(* IEC 61131-3 sources: AXOpen/src/components.festo.drives/app/src/IO, 10 files *)

(* ---- HwIdentifiers.st ---- *)
TYPE
	HwIdentifiers : ULINT
	(
		PLC_LINE_Rail_0 :=	ULINT#256,
		PLC_LINE_PLC_LINE :=	ULINT#48,
		PLC_LINE_Card_reader_writer_1 :=	ULINT#51,
		PLC_LINE_CPU_display_1 :=	ULINT#54,
		PLC_LINE_OPC_UA_1 :=	ULINT#117,
		PLC_LINE_PROFINET_interface_1 :=	ULINT#64,
		PLC_LINE_Port_1 :=	ULINT#65,
		PLC_LINE_Port_2 :=	ULINT#66,
		PLC_LINE_PROFINET_interface_2 :=	ULINT#72,
		PLC_LINE_DP_interface_1 :=	ULINT#60,
		PLC_LINE_PROFINET_interface_GBIT_3 :=	ULINT#120,
		ST3_indradrive_Rack :=	ULINT#336,
		ST3_indradrive_ST3_indradrive :=	ULINT#337,
		ST3_indradrive_PN_IO :=	ULINT#338,
		ST3_indradrive_Port_1_RJ45 :=	ULINT#339,
		ST3_indradrive_Port_2_RJ45 :=	ULINT#340,
		ST3_indradrive_DAP_1 :=	ULINT#341,
		ST3_indradrive_ID_FMod_NotUsed :=	ULINT#342,
		ST3_indradrive_ID_PaCh_5Words :=	ULINT#258,
		ST3_indradrive_ID_InMod_9Words :=	ULINT#262,
		ST3_indradrive_ID_OutMod_13Words :=	ULINT#259,
		cmmtas_PN_IO_Interface :=	ULINT#271,
		cmmtas_Port_1 :=	ULINT#260,
		cmmtas_Port_2 :=	ULINT#261,
		cmmtas_CMMT_AS_MP :=	ULINT#272,
		cmmtas_Module_Access_Point :=	ULINT#264,
		cmmtas_Siemens_telegram_111_PZD_12_12 :=	ULINT#265,
		cmmtas_Siemens_telegram_750_PZD_4_1 :=	ULINT#266,
		NONE:= ULINT#0
	);
END_TYPE

(* ---- HwInputs.st ---- *)
TYPE
	HwInputs : STRUCT
		ST3_indradrive_ID_PaCh_5Words AT %B10 : ARRAY[0..9] OF BYTE;
		ST3_indradrive_ID_InMod_9Words AT %B20 : ARRAY[0..17] OF BYTE;
		cmmtas_DO_SERVO_1_Siemens_telegram_111_PZD_12_12 AT %B100 : ARRAY[0..23] OF BYTE;
		cmmtas_DO_SERVO_1_Siemens_telegram_750_PZD_4_1 AT %B124 : WORD;
	END_STRUCT;
END_TYPE

(* ---- HwOutputs.st ---- *)
TYPE
	HwOutputs : STRUCT
		ST3_indradrive_ID_PaCh_5Words AT %B10 : ARRAY[0..9] OF BYTE;
		ST3_indradrive_ID_OutMod_13Words AT %B20 : ARRAY[0..25] OF BYTE;
		cmmtas_DO_SERVO_1_Siemens_telegram_111_PZD_12_12 AT %B100 : ARRAY[0..23] OF BYTE;
		cmmtas_DO_SERVO_1_Siemens_telegram_750_PZD_4_1 AT %B124 : ARRAY[0..7] OF BYTE;
	END_STRUCT;
END_TYPE

(* ---- Inputs.st ---- *)
NAMESPACE AXOpen.Components.Festo.Drives
    TYPE
        {S7.extern=ReadWrite}
        {#ix-attr:[Container(Layout.Wrap)]}
        Inputs : STRUCT
	        // Module festo_cmmtas/DoServo
	        festo_cmmtas_DoServo_SiemensTelegram111_PZD_12_12_Input AT %B0 : festo_cmmtas_DoServo_SiemensTelegram111_PZD_12_12_Input_Layout;

	        festo_cmmtas_DoServo_SiemensTelegram750_PZD_4_1_Input AT %B24 : festo_cmmtas_DoServo_SiemensTelegram750_PZD_4_1_Input_Layout;

        END_STRUCT;
    END_TYPE
END_NAMESPACE

(* ---- IoStructures.st ---- *)
NAMESPACE AXOpen.Components.Festo.Drives
	TYPE
        {S7.extern=ReadWrite}
        {#ix-attr:[Container(Layout.Wrap)]}
	    festo_cmmtas_DoServo_SiemensTelegram111_PZD_12_12_Input_Layout : STRUCT
	        Signals_0 AT %X0.0 : BOOL;
	        Signals_1 AT %X0.1 : BOOL;
	        Signals_2 AT %X0.2 : BOOL;
	        Signals_3 AT %X0.3 : BOOL;
	        Signals_4 AT %X0.4 : BOOL;
	        Signals_5 AT %X0.5 : BOOL;
	        Signals_6 AT %X0.6 : BOOL;
	        Signals_7 AT %X0.7 : BOOL;
	        Signals_8 AT %X1.0 : BOOL;
	        Signals_9 AT %X1.1 : BOOL;
	        Signals_10 AT %X1.2 : BOOL;
	        Signals_11 AT %X1.3 : BOOL;
	        Signals_12 AT %X1.4 : BOOL;
	        Signals_13 AT %X1.5 : BOOL;
	        Signals_14 AT %X1.6 : BOOL;
	        Signals_15 AT %X1.7 : BOOL;
	        Signals_16 AT %X2.0 : BOOL;
	        Signals_17 AT %X2.1 : BOOL;
	        Signals_18 AT %X2.2 : BOOL;
	        Signals_19 AT %X2.3 : BOOL;
	        Signals_20 AT %X2.4 : BOOL;
	        Signals_21 AT %X2.5 : BOOL;
	        Signals_22 AT %X2.6 : BOOL;
	        Signals_23 AT %X2.7 : BOOL;
	        Signals_24 AT %X3.0 : BOOL;
	        Signals_25 AT %X3.1 : BOOL;
	        Signals_26 AT %X3.2 : BOOL;
	        Signals_27 AT %X3.3 : BOOL;
	        Signals_28 AT %X3.4 : BOOL;
	        Signals_29 AT %X3.5 : BOOL;
	        Signals_30 AT %X3.6 : BOOL;
	        Signals_31 AT %X3.7 : BOOL;
	        Signals_32 AT %X4.0 : BOOL;
	        Signals_33 AT %X4.1 : BOOL;
	        Signals_34 AT %X4.2 : BOOL;
	        Signals_35 AT %X4.3 : BOOL;
	        Signals_36 AT %X4.4 : BOOL;
	        Signals_37 AT %X4.5 : BOOL;
	        Signals_38 AT %X4.6 : BOOL;
	        Signals_39 AT %X4.7 : BOOL;
	        Signals_40 AT %X5.0 : BOOL;
	        Signals_41 AT %X5.1 : BOOL;
	        Signals_42 AT %X5.2 : BOOL;
	        Signals_43 AT %X5.3 : BOOL;
	        Signals_44 AT %X5.4 : BOOL;
	        Signals_45 AT %X5.5 : BOOL;
	        Signals_46 AT %X5.6 : BOOL;
	        Signals_47 AT %X5.7 : BOOL;
	        Signals_48 AT %X6.0 : BOOL;
	        Signals_49 AT %X6.1 : BOOL;
	        Signals_50 AT %X6.2 : BOOL;
	        Signals_51 AT %X6.3 : BOOL;
	        Signals_52 AT %X6.4 : BOOL;
	        Signals_53 AT %X6.5 : BOOL;
	        Signals_54 AT %X6.6 : BOOL;
	        Signals_55 AT %X6.7 : BOOL;
	        Signals_56 AT %X7.0 : BOOL;
	        Signals_57 AT %X7.1 : BOOL;
	        Signals_58 AT %X7.2 : BOOL;
	        Signals_59 AT %X7.3 : BOOL;
	        Signals_60 AT %X7.4 : BOOL;
	        Signals_61 AT %X7.5 : BOOL;
	        Signals_62 AT %X7.6 : BOOL;
	        Signals_63 AT %X7.7 : BOOL;
	        Signals_64 AT %X8.0 : BOOL;
	        Signals_65 AT %X8.1 : BOOL;
	        Signals_66 AT %X8.2 : BOOL;
	        Signals_67 AT %X8.3 : BOOL;
	        Signals_68 AT %X8.4 : BOOL;
	        Signals_69 AT %X8.5 : BOOL;
	        Signals_70 AT %X8.6 : BOOL;
	        Signals_71 AT %X8.7 : BOOL;
	        Signals_72 AT %X9.0 : BOOL;
	        Signals_73 AT %X9.1 : BOOL;
	        Signals_74 AT %X9.2 : BOOL;
	        Signals_75 AT %X9.3 : BOOL;
	        Signals_76 AT %X9.4 : BOOL;
	        Signals_77 AT %X9.5 : BOOL;
	        Signals_78 AT %X9.6 : BOOL;
	        Signals_79 AT %X9.7 : BOOL;
	        Signals_80 AT %B10 : DWORD;
	        Signals_81 AT %B14 : DWORD;
	        Signals_82 AT %B18 : WORD;
	        Signals_83 AT %B20 : WORD;
	        Signals_84 AT %B22 : WORD;
	    END_STRUCT;
	END_TYPE

	TYPE
        {S7.extern=ReadWrite}
        {#ix-attr:[Container(Layout.Wrap)]}
	    festo_cmmtas_DoServo_SiemensTelegram111_PZD_12_12_Output_Layout : STRUCT
	        Signals_85 AT %X0.0 : BOOL;
	        Signals_86 AT %X0.1 : BOOL;
	        Signals_87 AT %X0.2 : BOOL;
	        Signals_88 AT %X0.3 : BOOL;
	        Signals_89 AT %X0.4 : BOOL;
	        Signals_90 AT %X0.5 : BOOL;
	        Signals_91 AT %X0.6 : BOOL;
	        Signals_92 AT %X0.7 : BOOL;
	        Signals_93 AT %X1.0 : BOOL;
	        Signals_94 AT %X1.1 : BOOL;
	        Signals_95 AT %X1.2 : BOOL;
	        Signals_96 AT %X1.3 : BOOL;
	        Signals_97 AT %X1.4 : BOOL;
	        Signals_98 AT %X1.5 : BOOL;
	        Signals_99 AT %X1.6 : BOOL;
	        Signals_100 AT %X1.7 : BOOL;
	        Signals_101 AT %X2.0 : BOOL;
	        Signals_102 AT %X2.1 : BOOL;
	        Signals_103 AT %X2.2 : BOOL;
	        Signals_104 AT %X2.3 : BOOL;
	        Signals_105 AT %X2.4 : BOOL;
	        Signals_106 AT %X2.5 : BOOL;
	        Signals_107 AT %X2.6 : BOOL;
	        Signals_108 AT %X2.7 : BOOL;
	        Signals_109 AT %X3.0 : BOOL;
	        Signals_110 AT %X3.1 : BOOL;
	        Signals_111 AT %X3.2 : BOOL;
	        Signals_112 AT %X3.3 : BOOL;
	        Signals_113 AT %X3.4 : BOOL;
	        Signals_114 AT %X3.5 : BOOL;
	        Signals_115 AT %X3.6 : BOOL;
	        Signals_116 AT %X3.7 : BOOL;
	        Signals_117 AT %X4.0 : BOOL;
	        Signals_118 AT %X4.1 : BOOL;
	        Signals_119 AT %X4.2 : BOOL;
	        Signals_120 AT %X4.3 : BOOL;
	        Signals_121 AT %X4.4 : BOOL;
	        Signals_122 AT %X4.5 : BOOL;
	        Signals_123 AT %X4.6 : BOOL;
	        Signals_124 AT %X4.7 : BOOL;
	        Signals_125 AT %X5.0 : BOOL;
	        Signals_126 AT %X5.1 : BOOL;
	        Signals_127 AT %X5.2 : BOOL;
	        Signals_128 AT %X5.3 : BOOL;
	        Signals_129 AT %X5.4 : BOOL;
	        Signals_130 AT %X5.5 : BOOL;
	        Signals_131 AT %X5.6 : BOOL;
	        Signals_132 AT %X5.7 : BOOL;
	        Signals_133 AT %X6.0 : BOOL;
	        Signals_134 AT %X6.1 : BOOL;
	        Signals_135 AT %X6.2 : BOOL;
	        Signals_136 AT %X6.3 : BOOL;
	        Signals_137 AT %X6.4 : BOOL;
	        Signals_138 AT %X6.5 : BOOL;
	        Signals_139 AT %X6.6 : BOOL;
	        Signals_140 AT %X6.7 : BOOL;
	        Signals_141 AT %X7.0 : BOOL;
	        Signals_142 AT %X7.1 : BOOL;
	        Signals_143 AT %X7.2 : BOOL;
	        Signals_144 AT %X7.3 : BOOL;
	        Signals_145 AT %X7.4 : BOOL;
	        Signals_146 AT %X7.5 : BOOL;
	        Signals_147 AT %X7.6 : BOOL;
	        Signals_148 AT %X7.7 : BOOL;
	        Signals_149 AT %B8 : WORD;
	        Signals_150 AT %B10 : DINT;
	        Signals_151 AT %B14 : DWORD;
	        Signals_152 AT %B18 : WORD;
	        Signals_153 AT %B20 : WORD;
	        Signals_154 AT %B22 : WORD;
	    END_STRUCT;
	END_TYPE

	TYPE
        {S7.extern=ReadWrite}
        {#ix-attr:[Container(Layout.Wrap)]}
	    festo_cmmtas_DoServo_SiemensTelegram750_PZD_4_1_Input_Layout : STRUCT
	        Signals_0 AT %B0 : WORD;
	    END_STRUCT;
	END_TYPE

	TYPE
        {S7.extern=ReadWrite}
        {#ix-attr:[Container(Layout.Wrap)]}
	    festo_cmmtas_DoServo_SiemensTelegram750_PZD_4_1_Output_Layout : STRUCT
	        Signals_1 AT %B0 : WORD;
	        Signals_2 AT %B2 : WORD;
	        Signals_3 AT %B4 : WORD;
	        Signals_4 AT %B6 : WORD;
	    END_STRUCT;
	END_TYPE
END_NAMESPACE

(* ---- Outputs.st ---- *)
NAMESPACE AXOpen.Components.Festo.Drives
    TYPE
        {S7.extern=ReadWrite}
        {#ix-attr:[Container(Layout.Wrap)]}
        Outputs : STRUCT
            cmmtas_DoServo_Submodule_1_0 AT %B0:  LWORD;
            cmmtas_DoServo_Submodule_1_1 AT %B8:  LWORD;
            cmmtas_DoServo_Submodule_1_2 AT %B16:  LWORD;
            cmmtas_DoServo_Submodule_2 AT %B24:  LWORD;
        END_STRUCT;
    END_TYPE
END_NAMESPACE

(* ---- PlcInputs.st ---- *)
TYPE
	PlcInputs : STRUCT
		ST3_indradrive_ID_PaCh_5Words : ARRAY[0..9] OF BYTE;
		ST3_indradrive_ID_InMod_9Words : ARRAY[0..17] OF BYTE;
		cmmtas_DO_SERVO_1_Siemens_telegram_111_PZD_12_12 : ARRAY[0..23] OF BYTE;
		cmmtas_DO_SERVO_1_Siemens_telegram_750_PZD_4_1 : WORD;
	END_STRUCT;
END_TYPE

(* ---- PlcOutputs.st ---- *)
TYPE
	PlcOutputs : STRUCT
		ST3_indradrive_ID_PaCh_5Words : ARRAY[0..9] OF BYTE;
		ST3_indradrive_ID_OutMod_13Words : ARRAY[0..25] OF BYTE;
		cmmtas_DO_SERVO_1_Siemens_telegram_111_PZD_12_12 : ARRAY[0..23] OF BYTE;
		cmmtas_DO_SERVO_1_Siemens_telegram_750_PZD_4_1 : ARRAY[0..7] OF BYTE;
	END_STRUCT;
END_TYPE

(* ---- CopyInputs.st ---- *)
FUNCTION CopyInputs
	VAR_EXTERNAL
		HwInputs : HwInputs;
		PlcInputs : PlcInputs;
	END_VAR
	PlcInputs.ST3_indradrive_ID_PaCh_5Words[0] := HwInputs.ST3_indradrive_ID_PaCh_5Words[0];
	PlcInputs.ST3_indradrive_ID_PaCh_5Words[1] := HwInputs.ST3_indradrive_ID_PaCh_5Words[1];
	PlcInputs.ST3_indradrive_ID_PaCh_5Words[2] := HwInputs.ST3_indradrive_ID_PaCh_5Words[2];
	PlcInputs.ST3_indradrive_ID_PaCh_5Words[3] := HwInputs.ST3_indradrive_ID_PaCh_5Words[3];
	PlcInputs.ST3_indradrive_ID_PaCh_5Words[4] := HwInputs.ST3_indradrive_ID_PaCh_5Words[4];
	PlcInputs.ST3_indradrive_ID_PaCh_5Words[5] := HwInputs.ST3_indradrive_ID_PaCh_5Words[5];
	PlcInputs.ST3_indradrive_ID_PaCh_5Words[6] := HwInputs.ST3_indradrive_ID_PaCh_5Words[6];
	PlcInputs.ST3_indradrive_ID_PaCh_5Words[7] := HwInputs.ST3_indradrive_ID_PaCh_5Words[7];
	PlcInputs.ST3_indradrive_ID_PaCh_5Words[8] := HwInputs.ST3_indradrive_ID_PaCh_5Words[8];
	PlcInputs.ST3_indradrive_ID_PaCh_5Words[9] := HwInputs.ST3_indradrive_ID_PaCh_5Words[9];
	PlcInputs.ST3_indradrive_ID_InMod_9Words[0] := HwInputs.ST3_indradrive_ID_InMod_9Words[0];
	PlcInputs.ST3_indradrive_ID_InMod_9Words[1] := HwInputs.ST3_indradrive_ID_InMod_9Words[1];
	PlcInputs.ST3_indradrive_ID_InMod_9Words[2] := HwInputs.ST3_indradrive_ID_InMod_9Words[2];
	PlcInputs.ST3_indradrive_ID_InMod_9Words[3] := HwInputs.ST3_indradrive_ID_InMod_9Words[3];
	PlcInputs.ST3_indradrive_ID_InMod_9Words[4] := HwInputs.ST3_indradrive_ID_InMod_9Words[4];
	PlcInputs.ST3_indradrive_ID_InMod_9Words[5] := HwInputs.ST3_indradrive_ID_InMod_9Words[5];
	PlcInputs.ST3_indradrive_ID_InMod_9Words[6] := HwInputs.ST3_indradrive_ID_InMod_9Words[6];
	PlcInputs.ST3_indradrive_ID_InMod_9Words[7] := HwInputs.ST3_indradrive_ID_InMod_9Words[7];
	PlcInputs.ST3_indradrive_ID_InMod_9Words[8] := HwInputs.ST3_indradrive_ID_InMod_9Words[8];
	PlcInputs.ST3_indradrive_ID_InMod_9Words[9] := HwInputs.ST3_indradrive_ID_InMod_9Words[9];
	PlcInputs.ST3_indradrive_ID_InMod_9Words[10] := HwInputs.ST3_indradrive_ID_InMod_9Words[10];
	PlcInputs.ST3_indradrive_ID_InMod_9Words[11] := HwInputs.ST3_indradrive_ID_InMod_9Words[11];
	PlcInputs.ST3_indradrive_ID_InMod_9Words[12] := HwInputs.ST3_indradrive_ID_InMod_9Words[12];
	PlcInputs.ST3_indradrive_ID_InMod_9Words[13] := HwInputs.ST3_indradrive_ID_InMod_9Words[13];
	PlcInputs.ST3_indradrive_ID_InMod_9Words[14] := HwInputs.ST3_indradrive_ID_InMod_9Words[14];
	PlcInputs.ST3_indradrive_ID_InMod_9Words[15] := HwInputs.ST3_indradrive_ID_InMod_9Words[15];
	PlcInputs.ST3_indradrive_ID_InMod_9Words[16] := HwInputs.ST3_indradrive_ID_InMod_9Words[16];
	PlcInputs.ST3_indradrive_ID_InMod_9Words[17] := HwInputs.ST3_indradrive_ID_InMod_9Words[17];
	PlcInputs.cmmtas_DO_SERVO_1_Siemens_telegram_111_PZD_12_12[0] := HwInputs.cmmtas_DO_SERVO_1_Siemens_telegram_111_PZD_12_12[0];
	PlcInputs.cmmtas_DO_SERVO_1_Siemens_telegram_111_PZD_12_12[1] := HwInputs.cmmtas_DO_SERVO_1_Siemens_telegram_111_PZD_12_12[1];
	PlcInputs.cmmtas_DO_SERVO_1_Siemens_telegram_111_PZD_12_12[2] := HwInputs.cmmtas_DO_SERVO_1_Siemens_telegram_111_PZD_12_12[2];
	PlcInputs.cmmtas_DO_SERVO_1_Siemens_telegram_111_PZD_12_12[3] := HwInputs.cmmtas_DO_SERVO_1_Siemens_telegram_111_PZD_12_12[3];
	PlcInputs.cmmtas_DO_SERVO_1_Siemens_telegram_111_PZD_12_12[4] := HwInputs.cmmtas_DO_SERVO_1_Siemens_telegram_111_PZD_12_12[4];
	PlcInputs.cmmtas_DO_SERVO_1_Siemens_telegram_111_PZD_12_12[5] := HwInputs.cmmtas_DO_SERVO_1_Siemens_telegram_111_PZD_12_12[5];
	PlcInputs.cmmtas_DO_SERVO_1_Siemens_telegram_111_PZD_12_12[6] := HwInputs.cmmtas_DO_SERVO_1_Siemens_telegram_111_PZD_12_12[6];
	PlcInputs.cmmtas_DO_SERVO_1_Siemens_telegram_111_PZD_12_12[7] := HwInputs.cmmtas_DO_SERVO_1_Siemens_telegram_111_PZD_12_12[7];
	PlcInputs.cmmtas_DO_SERVO_1_Siemens_telegram_111_PZD_12_12[8] := HwInputs.cmmtas_DO_SERVO_1_Siemens_telegram_111_PZD_12_12[8];
	PlcInputs.cmmtas_DO_SERVO_1_Siemens_telegram_111_PZD_12_12[9] := HwInputs.cmmtas_DO_SERVO_1_Siemens_telegram_111_PZD_12_12[9];
	PlcInputs.cmmtas_DO_SERVO_1_Siemens_telegram_111_PZD_12_12[10] := HwInputs.cmmtas_DO_SERVO_1_Siemens_telegram_111_PZD_12_12[10];
	PlcInputs.cmmtas_DO_SERVO_1_Siemens_telegram_111_PZD_12_12[11] := HwInputs.cmmtas_DO_SERVO_1_Siemens_telegram_111_PZD_12_12[11];
	PlcInputs.cmmtas_DO_SERVO_1_Siemens_telegram_111_PZD_12_12[12] := HwInputs.cmmtas_DO_SERVO_1_Siemens_telegram_111_PZD_12_12[12];
	PlcInputs.cmmtas_DO_SERVO_1_Siemens_telegram_111_PZD_12_12[13] := HwInputs.cmmtas_DO_SERVO_1_Siemens_telegram_111_PZD_12_12[13];
	PlcInputs.cmmtas_DO_SERVO_1_Siemens_telegram_111_PZD_12_12[14] := HwInputs.cmmtas_DO_SERVO_1_Siemens_telegram_111_PZD_12_12[14];
	PlcInputs.cmmtas_DO_SERVO_1_Siemens_telegram_111_PZD_12_12[15] := HwInputs.cmmtas_DO_SERVO_1_Siemens_telegram_111_PZD_12_12[15];
	PlcInputs.cmmtas_DO_SERVO_1_Siemens_telegram_111_PZD_12_12[16] := HwInputs.cmmtas_DO_SERVO_1_Siemens_telegram_111_PZD_12_12[16];
	PlcInputs.cmmtas_DO_SERVO_1_Siemens_telegram_111_PZD_12_12[17] := HwInputs.cmmtas_DO_SERVO_1_Siemens_telegram_111_PZD_12_12[17];
	PlcInputs.cmmtas_DO_SERVO_1_Siemens_telegram_111_PZD_12_12[18] := HwInputs.cmmtas_DO_SERVO_1_Siemens_telegram_111_PZD_12_12[18];
	PlcInputs.cmmtas_DO_SERVO_1_Siemens_telegram_111_PZD_12_12[19] := HwInputs.cmmtas_DO_SERVO_1_Siemens_telegram_111_PZD_12_12[19];
	PlcInputs.cmmtas_DO_SERVO_1_Siemens_telegram_111_PZD_12_12[20] := HwInputs.cmmtas_DO_SERVO_1_Siemens_telegram_111_PZD_12_12[20];
	PlcInputs.cmmtas_DO_SERVO_1_Siemens_telegram_111_PZD_12_12[21] := HwInputs.cmmtas_DO_SERVO_1_Siemens_telegram_111_PZD_12_12[21];
	PlcInputs.cmmtas_DO_SERVO_1_Siemens_telegram_111_PZD_12_12[22] := HwInputs.cmmtas_DO_SERVO_1_Siemens_telegram_111_PZD_12_12[22];
	PlcInputs.cmmtas_DO_SERVO_1_Siemens_telegram_111_PZD_12_12[23] := HwInputs.cmmtas_DO_SERVO_1_Siemens_telegram_111_PZD_12_12[23];
	PlcInputs.cmmtas_DO_SERVO_1_Siemens_telegram_750_PZD_4_1 := HwInputs.cmmtas_DO_SERVO_1_Siemens_telegram_750_PZD_4_1;
END_FUNCTION

(* ---- CopyOutputs.st ---- *)
FUNCTION CopyOutputs
	VAR_EXTERNAL
		HwOutputs : HwOutputs;
		PlcOutputs : PlcOutputs;
	END_VAR
	HwOutputs.ST3_indradrive_ID_PaCh_5Words[0] := PlcOutputs.ST3_indradrive_ID_PaCh_5Words[0];
	HwOutputs.ST3_indradrive_ID_PaCh_5Words[1] := PlcOutputs.ST3_indradrive_ID_PaCh_5Words[1];
	HwOutputs.ST3_indradrive_ID_PaCh_5Words[2] := PlcOutputs.ST3_indradrive_ID_PaCh_5Words[2];
	HwOutputs.ST3_indradrive_ID_PaCh_5Words[3] := PlcOutputs.ST3_indradrive_ID_PaCh_5Words[3];
	HwOutputs.ST3_indradrive_ID_PaCh_5Words[4] := PlcOutputs.ST3_indradrive_ID_PaCh_5Words[4];
	HwOutputs.ST3_indradrive_ID_PaCh_5Words[5] := PlcOutputs.ST3_indradrive_ID_PaCh_5Words[5];
	HwOutputs.ST3_indradrive_ID_PaCh_5Words[6] := PlcOutputs.ST3_indradrive_ID_PaCh_5Words[6];
	HwOutputs.ST3_indradrive_ID_PaCh_5Words[7] := PlcOutputs.ST3_indradrive_ID_PaCh_5Words[7];
	HwOutputs.ST3_indradrive_ID_PaCh_5Words[8] := PlcOutputs.ST3_indradrive_ID_PaCh_5Words[8];
	HwOutputs.ST3_indradrive_ID_PaCh_5Words[9] := PlcOutputs.ST3_indradrive_ID_PaCh_5Words[9];
	HwOutputs.ST3_indradrive_ID_OutMod_13Words[0] := PlcOutputs.ST3_indradrive_ID_OutMod_13Words[0];
	HwOutputs.ST3_indradrive_ID_OutMod_13Words[1] := PlcOutputs.ST3_indradrive_ID_OutMod_13Words[1];
	HwOutputs.ST3_indradrive_ID_OutMod_13Words[2] := PlcOutputs.ST3_indradrive_ID_OutMod_13Words[2];
	HwOutputs.ST3_indradrive_ID_OutMod_13Words[3] := PlcOutputs.ST3_indradrive_ID_OutMod_13Words[3];
	HwOutputs.ST3_indradrive_ID_OutMod_13Words[4] := PlcOutputs.ST3_indradrive_ID_OutMod_13Words[4];
	HwOutputs.ST3_indradrive_ID_OutMod_13Words[5] := PlcOutputs.ST3_indradrive_ID_OutMod_13Words[5];
	HwOutputs.ST3_indradrive_ID_OutMod_13Words[6] := PlcOutputs.ST3_indradrive_ID_OutMod_13Words[6];
	HwOutputs.ST3_indradrive_ID_OutMod_13Words[7] := PlcOutputs.ST3_indradrive_ID_OutMod_13Words[7];
	HwOutputs.ST3_indradrive_ID_OutMod_13Words[8] := PlcOutputs.ST3_indradrive_ID_OutMod_13Words[8];
	HwOutputs.ST3_indradrive_ID_OutMod_13Words[9] := PlcOutputs.ST3_indradrive_ID_OutMod_13Words[9];
	HwOutputs.ST3_indradrive_ID_OutMod_13Words[10] := PlcOutputs.ST3_indradrive_ID_OutMod_13Words[10];
	HwOutputs.ST3_indradrive_ID_OutMod_13Words[11] := PlcOutputs.ST3_indradrive_ID_OutMod_13Words[11];
	HwOutputs.ST3_indradrive_ID_OutMod_13Words[12] := PlcOutputs.ST3_indradrive_ID_OutMod_13Words[12];
	HwOutputs.ST3_indradrive_ID_OutMod_13Words[13] := PlcOutputs.ST3_indradrive_ID_OutMod_13Words[13];
	HwOutputs.ST3_indradrive_ID_OutMod_13Words[14] := PlcOutputs.ST3_indradrive_ID_OutMod_13Words[14];
	HwOutputs.ST3_indradrive_ID_OutMod_13Words[15] := PlcOutputs.ST3_indradrive_ID_OutMod_13Words[15];
	HwOutputs.ST3_indradrive_ID_OutMod_13Words[16] := PlcOutputs.ST3_indradrive_ID_OutMod_13Words[16];
	HwOutputs.ST3_indradrive_ID_OutMod_13Words[17] := PlcOutputs.ST3_indradrive_ID_OutMod_13Words[17];
	HwOutputs.ST3_indradrive_ID_OutMod_13Words[18] := PlcOutputs.ST3_indradrive_ID_OutMod_13Words[18];
	HwOutputs.ST3_indradrive_ID_OutMod_13Words[19] := PlcOutputs.ST3_indradrive_ID_OutMod_13Words[19];
	HwOutputs.ST3_indradrive_ID_OutMod_13Words[20] := PlcOutputs.ST3_indradrive_ID_OutMod_13Words[20];
	HwOutputs.ST3_indradrive_ID_OutMod_13Words[21] := PlcOutputs.ST3_indradrive_ID_OutMod_13Words[21];
	HwOutputs.ST3_indradrive_ID_OutMod_13Words[22] := PlcOutputs.ST3_indradrive_ID_OutMod_13Words[22];
	HwOutputs.ST3_indradrive_ID_OutMod_13Words[23] := PlcOutputs.ST3_indradrive_ID_OutMod_13Words[23];
	HwOutputs.ST3_indradrive_ID_OutMod_13Words[24] := PlcOutputs.ST3_indradrive_ID_OutMod_13Words[24];
	HwOutputs.ST3_indradrive_ID_OutMod_13Words[25] := PlcOutputs.ST3_indradrive_ID_OutMod_13Words[25];
	HwOutputs.cmmtas_DO_SERVO_1_Siemens_telegram_111_PZD_12_12[0] := PlcOutputs.cmmtas_DO_SERVO_1_Siemens_telegram_111_PZD_12_12[0];
	HwOutputs.cmmtas_DO_SERVO_1_Siemens_telegram_111_PZD_12_12[1] := PlcOutputs.cmmtas_DO_SERVO_1_Siemens_telegram_111_PZD_12_12[1];
	HwOutputs.cmmtas_DO_SERVO_1_Siemens_telegram_111_PZD_12_12[2] := PlcOutputs.cmmtas_DO_SERVO_1_Siemens_telegram_111_PZD_12_12[2];
	HwOutputs.cmmtas_DO_SERVO_1_Siemens_telegram_111_PZD_12_12[3] := PlcOutputs.cmmtas_DO_SERVO_1_Siemens_telegram_111_PZD_12_12[3];
	HwOutputs.cmmtas_DO_SERVO_1_Siemens_telegram_111_PZD_12_12[4] := PlcOutputs.cmmtas_DO_SERVO_1_Siemens_telegram_111_PZD_12_12[4];
	HwOutputs.cmmtas_DO_SERVO_1_Siemens_telegram_111_PZD_12_12[5] := PlcOutputs.cmmtas_DO_SERVO_1_Siemens_telegram_111_PZD_12_12[5];
	HwOutputs.cmmtas_DO_SERVO_1_Siemens_telegram_111_PZD_12_12[6] := PlcOutputs.cmmtas_DO_SERVO_1_Siemens_telegram_111_PZD_12_12[6];
	HwOutputs.cmmtas_DO_SERVO_1_Siemens_telegram_111_PZD_12_12[7] := PlcOutputs.cmmtas_DO_SERVO_1_Siemens_telegram_111_PZD_12_12[7];
	HwOutputs.cmmtas_DO_SERVO_1_Siemens_telegram_111_PZD_12_12[8] := PlcOutputs.cmmtas_DO_SERVO_1_Siemens_telegram_111_PZD_12_12[8];
	HwOutputs.cmmtas_DO_SERVO_1_Siemens_telegram_111_PZD_12_12[9] := PlcOutputs.cmmtas_DO_SERVO_1_Siemens_telegram_111_PZD_12_12[9];
	HwOutputs.cmmtas_DO_SERVO_1_Siemens_telegram_111_PZD_12_12[10] := PlcOutputs.cmmtas_DO_SERVO_1_Siemens_telegram_111_PZD_12_12[10];
	HwOutputs.cmmtas_DO_SERVO_1_Siemens_telegram_111_PZD_12_12[11] := PlcOutputs.cmmtas_DO_SERVO_1_Siemens_telegram_111_PZD_12_12[11];
	HwOutputs.cmmtas_DO_SERVO_1_Siemens_telegram_111_PZD_12_12[12] := PlcOutputs.cmmtas_DO_SERVO_1_Siemens_telegram_111_PZD_12_12[12];
	HwOutputs.cmmtas_DO_SERVO_1_Siemens_telegram_111_PZD_12_12[13] := PlcOutputs.cmmtas_DO_SERVO_1_Siemens_telegram_111_PZD_12_12[13];
	HwOutputs.cmmtas_DO_SERVO_1_Siemens_telegram_111_PZD_12_12[14] := PlcOutputs.cmmtas_DO_SERVO_1_Siemens_telegram_111_PZD_12_12[14];
	HwOutputs.cmmtas_DO_SERVO_1_Siemens_telegram_111_PZD_12_12[15] := PlcOutputs.cmmtas_DO_SERVO_1_Siemens_telegram_111_PZD_12_12[15];
	HwOutputs.cmmtas_DO_SERVO_1_Siemens_telegram_111_PZD_12_12[16] := PlcOutputs.cmmtas_DO_SERVO_1_Siemens_telegram_111_PZD_12_12[16];
	HwOutputs.cmmtas_DO_SERVO_1_Siemens_telegram_111_PZD_12_12[17] := PlcOutputs.cmmtas_DO_SERVO_1_Siemens_telegram_111_PZD_12_12[17];
	HwOutputs.cmmtas_DO_SERVO_1_Siemens_telegram_111_PZD_12_12[18] := PlcOutputs.cmmtas_DO_SERVO_1_Siemens_telegram_111_PZD_12_12[18];
	HwOutputs.cmmtas_DO_SERVO_1_Siemens_telegram_111_PZD_12_12[19] := PlcOutputs.cmmtas_DO_SERVO_1_Siemens_telegram_111_PZD_12_12[19];
	HwOutputs.cmmtas_DO_SERVO_1_Siemens_telegram_111_PZD_12_12[20] := PlcOutputs.cmmtas_DO_SERVO_1_Siemens_telegram_111_PZD_12_12[20];
	HwOutputs.cmmtas_DO_SERVO_1_Siemens_telegram_111_PZD_12_12[21] := PlcOutputs.cmmtas_DO_SERVO_1_Siemens_telegram_111_PZD_12_12[21];
	HwOutputs.cmmtas_DO_SERVO_1_Siemens_telegram_111_PZD_12_12[22] := PlcOutputs.cmmtas_DO_SERVO_1_Siemens_telegram_111_PZD_12_12[22];
	HwOutputs.cmmtas_DO_SERVO_1_Siemens_telegram_111_PZD_12_12[23] := PlcOutputs.cmmtas_DO_SERVO_1_Siemens_telegram_111_PZD_12_12[23];
	HwOutputs.cmmtas_DO_SERVO_1_Siemens_telegram_750_PZD_4_1[0] := PlcOutputs.cmmtas_DO_SERVO_1_Siemens_telegram_750_PZD_4_1[0];
	HwOutputs.cmmtas_DO_SERVO_1_Siemens_telegram_750_PZD_4_1[1] := PlcOutputs.cmmtas_DO_SERVO_1_Siemens_telegram_750_PZD_4_1[1];
	HwOutputs.cmmtas_DO_SERVO_1_Siemens_telegram_750_PZD_4_1[2] := PlcOutputs.cmmtas_DO_SERVO_1_Siemens_telegram_750_PZD_4_1[2];
	HwOutputs.cmmtas_DO_SERVO_1_Siemens_telegram_750_PZD_4_1[3] := PlcOutputs.cmmtas_DO_SERVO_1_Siemens_telegram_750_PZD_4_1[3];
	HwOutputs.cmmtas_DO_SERVO_1_Siemens_telegram_750_PZD_4_1[4] := PlcOutputs.cmmtas_DO_SERVO_1_Siemens_telegram_750_PZD_4_1[4];
	HwOutputs.cmmtas_DO_SERVO_1_Siemens_telegram_750_PZD_4_1[5] := PlcOutputs.cmmtas_DO_SERVO_1_Siemens_telegram_750_PZD_4_1[5];
	HwOutputs.cmmtas_DO_SERVO_1_Siemens_telegram_750_PZD_4_1[6] := PlcOutputs.cmmtas_DO_SERVO_1_Siemens_telegram_750_PZD_4_1[6];
	HwOutputs.cmmtas_DO_SERVO_1_Siemens_telegram_750_PZD_4_1[7] := PlcOutputs.cmmtas_DO_SERVO_1_Siemens_telegram_750_PZD_4_1[7];
END_FUNCTION
